// TIA Portal V17 export
// export: Created 2025-06-26T06:49:22.0519669Z, ExportSetting WithDefaults, DisplayName Totally Integrated Automation Portal, DisplayVersion V17 Update 8, DisplayName TIA Portal Openness, DisplayVersion V17 Update 8, DisplayName TIA Portal Version Control Interface, DisplayVersion V17, DisplayName STEP 7 Professional, DisplayVersion V17 Update 8, DisplayName STEP 7 Safety, DisplayVersion V17 Update 6, DisplayName WinCC Advanced, DisplayVersion V17 Update 8
DATA_BLOCK "DB_TestSupport"   // DB6
{ S7_Optimized_Access := 'TRUE' }
VERSION : 0.1
// stored: AutoNumber true, DBAccessibleFromOPCUA true, IsOnlyStoredInLoadMemory false, IsRetainMemResEnabled false, IsWriteProtectedInAS false, MemoryReserve 100
   VAR
      AI : Struct
         TSS_TT_201 { S7_SetPoint := 'True'} : "stCalcValue";   // Heat source tank temperature
         TSS_TT_202 { S7_SetPoint := 'True'} : "stCalcValue";   // Heat sink tank temperature
         TSS_TT_206 { S7_SetPoint := 'True'} : "stCalcValue";   // Heat source suction temperature
         TSS_TT_208 { S7_SetPoint := 'True'} : "stCalcValue";   // Heat sink suction temperature
         TSS_TT_209 { S7_SetPoint := 'True'} : "stCalcValue";   // Heat sink discharge temperature
         TSS_FT_210 { S7_SetPoint := 'True'} : "stCalcValue";   // Heat source flow
         TSS_FT_211 { S7_SetPoint := 'True'} : "stCalcValue";   // Heat sink flow
         TSS_SC_213 { S7_SetPoint := 'True'} : "stCalcValue";   // Heat source feed pump speed
         TSS_SC_214 { S7_SetPoint := 'True'} : "stCalcValue";   // Heat sink feed pump speed
         TSA_PT_300 { S7_SetPoint := 'True'} : "stCalcValue";   // Heat sink cycle condensate pump suction pressure
         TSA_TT_301 { S7_SetPoint := 'True'} : "stCalcValue";   // Heat sink cycle condensate pump suction temperature
         TSA_TT_304 { S7_SetPoint := 'True'} : "stCalcValue";   // Heat sink cycle condensate tank suction temperature
         TSA_PT_306 { S7_SetPoint := 'True'} : "stCalcValue";   // Heat sink cycle condensate pump discharge pressure
         TSA_FT_307 { S7_SetPoint := 'True'} : "stCalcValue";   // Heat sink cycle condensate pump discharge flow
         TSA_LT_308 { S7_SetPoint := 'True'} : "stCalcValue";   // Heat sink cycle condensate tank level
         TSA_TT_320 { S7_SetPoint := 'True'} : "stCalcValue";   // Steam generator discharge temperature
         TSA_PT_321 { S7_SetPoint := 'True'} : "stCalcValue";   // Steam generator discharge pressure
         TSA_PT_323 { S7_SetPoint := 'True'} : "stCalcValue";   // Steam system pressure (?)
         TSA_TT_324 { S7_SetPoint := 'True'} : "stCalcValue";   // Steam system temperature (?)
         TSA_PT_328 { S7_SetPoint := 'True'} : "stCalcValue";   // Nitrogen blanketing pressure
         TSA_PT_350 { S7_SetPoint := 'True'} : "stCalcValue";   // Heat source cycle condensate pump suction pressure
         TSA_TT_351 { S7_SetPoint := 'True'} : "stCalcValue";   // Heat source cycle condensate pump suction temperature
         TSA_PT_354 { S7_SetPoint := 'True'} : "stCalcValue";   // Heat source cycle condensate pump discharge pressure
         TSA_FT_355 { S7_SetPoint := 'True'} : "stCalcValue";   // Heat source cycle condensate pump discharge flow
         TSA_TT_356 { S7_SetPoint := 'True'} : "stCalcValue";   // Heat source suction temperature
         TSA_PT_374 { S7_SetPoint := 'True'} : "stCalcValue";   // Heat source suction pressure
      END_STRUCT;
      DI : Struct
         TSA_HV_326 : Bool;   // Heat sink cycle nitrogen blanketing valve 1
         TSA_HV_327 : Bool;   // Heat sink cycle nitrogen blanketing valve 2
         TSA_HV_330 : Bool;   // Preheating pump discharge valve
         TSA_HV_372 : Bool;   // Heat source cycle nitrogen blanketing valve 1
         TSA_HV_373 : Bool;   // Heat source cycle nitrogen blanketing valve 2
         Spare05 : Bool;
         Spare06 : Bool;
         Spare07 : Bool;
         Spare10 : Bool;
         Spare11 : Bool;
         Spare12 : Bool;
         Spare13 : Bool;
         Spare14 : Bool;
         Spare15 : Bool;
         Spare16 : Bool;
         Spare17 : Bool;
      END_STRUCT;
      Valve : Struct
         TSS_HCV_301_A1 { S7_SetPoint := 'True'} : "stCalcValue";   // Heat source 3-way mix valve position
         TSS_HCV_302_A1 { S7_SetPoint := 'True'} : "stCalcValue";   // Heat sink 3-way mix valve position
         TSA_HCV_322_A1 { S7_SetPoint := 'True'} : "stCalcValue";   // Heat sink cycle control valve position
         TSA_HCV_370_A1 { S7_SetPoint := 'True'} : "stCalcValue";   // Heat source cycle control valve position
      END_STRUCT;
      Inverter : Struct
         TSA_SC_301 : "stCalcValue";
         TSA_SC_330 : "stCalcValue";
         TSA_SC_351 : "stCalcValue";
      END_STRUCT;
   END_VAR
BEGIN
END_DATA_BLOCK
